// TIA Portal V20 export
// export: Created 2025-12-01T14:57:41.2764139Z, ExportSetting None, DisplayName Totally Integrated Automation Portal, DisplayVersion V20 Update 3, DisplayName TIA Portal Openness, DisplayVersion V20 Update 3, DisplayName TIA Portal Version Control Interface, DisplayVersion V20 Update 3, DisplayName STEP 7 Professional, DisplayVersion V20 Update 3, DisplayName STEP 7 Safety, DisplayVersion V20 Update 2, DisplayName WinCC Basic/Comfort/Advanced, DisplayVersion V20 Update 3, DisplayName WinCC Professional, DisplayVersion V20 Update 3, DisplayName WinCC Unified, DisplayVersion V20 Update 3
FUNCTION "FC973_HMI_NDD" : Void   // FC973, LAD
{ S7_Optimized_Access := 'FALSE' }
// stored: AutoNumber false, SetENOAutomatically false
   VAR_INPUT
      DirEntradas : UInt;
      DiRSalidas : UInt;
      DirEntradasSeguras : UInt;
      DirSalidasSeguras : UInt;
      ElevadorPosicion : Int;
      HorquillaPosicion : Int;
      GarraPosicion : Int;
      ElevadorReferenciaOK : Bool;
      HorquillaReferenciaOK : Bool;
      GarraReferenciaOK : Bool;
   END_VAR
   VAR_IN_OUT
      HMI : "NDD_HMI";
   END_VAR
   VAR_TEMP
      Guardar_AR2 : DWord;
      P_Any : Any;
      LongEntradas : UInt;
      LongSalidas : UInt;
      LongEntradasSeguras : UInt;
      LongSalidasSeguras : UInt;
      ReturnValor : Int;
   END_VAR
BEGIN

NETWORK
TITLE = Inicializar
///////////////////////////////////////////////////////////////////////////////////////
/// Longitudes de las Entradas y Salidas - Normales

      L     14;
      T     #LongEntradas;
      L     4;
      T     #LongSalidas;


///////////////////////////////////////////////////////////////////////////////////////
/// Longitudes de las Entradas y Salidas - Seguras

      L     6;
      T     #LongEntradasSeguras;
      L     3;
      T     #LongSalidasSeguras;



NETWORK
TITLE = Copia de las Entradas Normales
///////////////////////////////////////////////////////////////////////////////////////
/// Preparar el puntero ANY de las Entradas Normales

      TAR2  #Guardar_AR2;  // Guardar AR2

      LAR2  P##P_Any;  // - Any - Entradas del interlock
      L     B#16#10;  //   10H para S7
      T     LB [AR2, P#0.0];
      L     B#16#2;  //   Tipo de Datos (BYTE)
      T     LB [AR2, P#1.0];
      L     #LongEntradas;  //   Cantidad de datos
      T     LW [AR2, P#2.0];
      L     0;  //   Numero de DB (Temporal = 0)
      T     LW [AR2, P#4.0];
      L     #DirEntradas;  //   Direccion de Inicio
      SLD   3;
      T     LD [AR2, P#6.0];
      L     B#16#81;  //   El Area de Memoria = Entradas
      T     LB [AR2, P#6.0];

      LAR2  #Guardar_AR2;  // Recuperar AR2


/// Copiar las Entradas

      CALL  UBLKMOV
      ( SRCBLK  := #P_Any,
        RET_VAL := #ReturnValor,
        DSTBLK  := #HMI.Entradas
      );



NETWORK
TITLE = Copia de las Salidas Normales
///////////////////////////////////////////////////////////////////////////////////////
/// Preparar el puntero ANY de las Salidas Normales

      TAR2  #Guardar_AR2;  // Guardar AR2

      LAR2  P##P_Any;  // - Any - Entradas del interlock
      L     B#16#10;  //   10H para S7
      T     LB [AR2, P#0.0];
      L     B#16#2;  //   Tipo de Datos (BYTE)
      T     LB [AR2, P#1.0];
      L     #LongSalidas;  //   Cantidad de datos
      T     LW [AR2, P#2.0];
      L     0;  //   Numero de DB (Temporal = 0)
      T     LW [AR2, P#4.0];
      L     #DiRSalidas;  //   Direccion de Inicio
      SLD   3;
      T     LD [AR2, P#6.0];
      L     B#16#82;  //   El Area de Memoria = Entradas
      T     LB [AR2, P#6.0];

      LAR2  #Guardar_AR2;  // Recuperar AR2


/// Copiar las Entradas

      CALL  UBLKMOV
      ( SRCBLK  := #P_Any,
        RET_VAL := #ReturnValor,
        DSTBLK  := #HMI.Salidas
      );



NETWORK
TITLE = Copia de las Entradas Seguras
///////////////////////////////////////////////////////////////////////////////////////
/// Preparar el puntero ANY de las Entradas Normales

      TAR2  #Guardar_AR2;  // Guardar AR2

      LAR2  P##P_Any;  // - Any - Entradas del interlock
      L     B#16#10;  //   10H para S7
      T     LB [AR2, P#0.0];
      L     B#16#2;  //   Tipo de Datos (BYTE)
      T     LB [AR2, P#1.0];
      L     #LongEntradasSeguras;  //   Cantidad de datos
      L     6;  // Tamaño de la tarjeta segura
      *I;
      T     LW [AR2, P#2.0];
      L     0;  //   Numero de DB (Temporal = 0)
      T     LW [AR2, P#4.0];
      L     #DirEntradasSeguras;  //   Direccion de Inicio
      SLD   3;
      T     LD [AR2, P#6.0];
      L     B#16#81;  //   El Area de Memoria = Entradas
      T     LB [AR2, P#6.0];

      LAR2  #Guardar_AR2;  // Recuperar AR2


/// Copiar las Entradas

      CALL  UBLKMOV
      ( SRCBLK  := #P_Any,
        RET_VAL := #ReturnValor,
        DSTBLK  := #HMI.EntradasSeguras
      );



NETWORK
TITLE = Copia de las Salidas Seguras
///////////////////////////////////////////////////////////////////////////////////////
/// Preparar el puntero ANY de las Salidas Normales

      TAR2  #Guardar_AR2;  // Guardar AR2

      LAR2  P##P_Any;  // - Any - Entradas del interlock
      L     B#16#10;  //   10H para S7
      T     LB [AR2, P#0.0];
      L     B#16#2;  //   Tipo de Datos (BYTE)
      T     LB [AR2, P#1.0];
      L     #LongSalidasSeguras;  //   Cantidad de datos
      L     6;  // Tamaño de la tarjeta segura
      *I;
      T     LW [AR2, P#2.0];
      L     0;  //   Numero de DB (Temporal = 0)
      T     LW [AR2, P#4.0];
      L     #DirSalidasSeguras;  //   Direccion de Inicio
      SLD   3;
      T     LD [AR2, P#6.0];
      L     B#16#82;  //   El Area de Memoria = Entradas
      T     LB [AR2, P#6.0];

      LAR2  #Guardar_AR2;  // Recuperar AR2


/// Copiar las Entradas

      CALL  UBLKMOV
      ( SRCBLK  := #P_Any,
        RET_VAL := #ReturnValor,
        DSTBLK  := #HMI.SalidasSeguras
      );




NETWORK
TITLE = Datos del Elevador, Horquilla y Garra
///////////////////////////////////////////////////////////////////////////////////////
/// Datos del Elevador

      SET;
      A     #ElevadorReferenciaOK;
      =     #HMI.Elevador.ReferenciaOK;

      L     #ElevadorPosicion;
      T     #HMI.Elevador.Posicion;


///////////////////////////////////////////////////////////////////////////////////////
/// Datos de la Horquilla

      SET;
      A     #HorquillaReferenciaOK;
      =     #HMI.Horquilla.ReferenciaOK;

      L     #HorquillaPosicion;
      T     #HMI.Horquilla.Posicion;


///////////////////////////////////////////////////////////////////////////////////////
/// Datos de la Garra

      SET;
      A     #GarraReferenciaOK;
      =     #HMI.Garra.ReferenciaOK;

      L     #GarraPosicion;
      T     #HMI.Garra.Posicion;



NETWORK
TITLE = 
///////////////////////////////////////////////////////////////////////////////////////
///


END_FUNCTION
